{attribute 'GeneratedUsingTerminal: EK1122-0000-0018'}
{attribute addProperty BoxType "EK1122-0000-0018"}
{attribute addProperty Id "Beckhoff_EL25xxsub_EK1100EK1100_AB5A94672"}
{attribute addProperty CRC "1829665105"}
{attribute addProperty Size "2"}
TYPE Beckhoff_EL25xxEK1122_6D0E7951 EXTENDS EK1122_AB5A9467 :
STRUCT
	{attribute addProperty Name "Beckhoff_EL25xxsub_EK1100"}
	{attribute addProperty PreviousPort "Beckhoff EL25xxEK1122 : D"}
	Beckhoff_EL25xxsub_EK1100 : EK1100_AB5A9467;
END_STRUCT
END_TYPE

(* stored: Version 1.2.0.0, ProductVersion 3.1.4024.9
   DUT Beckhoff_EL25xxEK1122_6D0E7951: Id {23bcd79b-4696-4614-a3e8-df83669c9402} *)
